// TIA Portal V20 export
DATA_BLOCK "ShiftmodelInterfaceHmi"   // DB103
TITLE = Schichtzeiten / ShiftmodelTimes
AUTHOR : SICAR
FAMILY : Shiftmodel
VERSION : 1.0
// Global DB fuer Schnittstelle HMI / Global DB for HMI interface
// stored: InstanceOfName LSicar_typeShiftmodelHmi, InstanceOfType UDT
"LSicar_typeShiftmodelHmi"
   // VAR RETAIN
   //    shiftTimesListIndex : DInt := 1;
   //    actualTimesDay : Array[0..7] of "LSicar_typeShiftmodTime1Day";
   //    actualSignalsDay : Array[0..7] of "LSicar_typeShiftmodSign1Day";
   //    summary : "LSicar_typeShiftmodSumHmi";
   //    actualDay : USInt := 0;
   //    shiftTimesListOnOff : Bool := TRUE;   // Schichtzeiten Remote OnOff / Shift times OnOff
   //    setAdjTimes : Bool := FALSE;
   //    hmiTimesValidFor : Array[0..3] of "LSicar_typeWeekdayBools";
   //    hmiTimes : Array[0..3] of "LSicar_typeShiftmodTime1Shift";   // Schnittstelle Lokale Zeiten (eingeben am HMI) / Interface Local Times (Input on HMI)
   //    productionTimes : "LSicar_typeProdTimesHmi";
   // END_VAR
BEGIN
   actualTimesDay[0].shift[0..3].endCircuitTime := TOD#00:00:00;
   actualTimesDay[1].shift[0..3].endCircuitTime := TOD#00:00:00;
   actualTimesDay[2].shift[0..3].endCircuitTime := TOD#00:00:00;
   actualTimesDay[3].shift[0..3].endCircuitTime := TOD#00:00:00;
   actualTimesDay[4].shift[0..3].endCircuitTime := TOD#00:00:00;
   actualTimesDay[5].shift[0..3].endCircuitTime := TOD#00:00:00;
   actualTimesDay[6].shift[0..3].endCircuitTime := TOD#00:00:00;
   actualTimesDay[7].shift[0..3].endCircuitTime := TOD#00:00:00;
   actualTimesDay[0].shift[0..3].start := TOD#00:00:00;
   actualTimesDay[1].shift[0..3].start := TOD#00:00:00;
   actualTimesDay[2].shift[0..3].start := TOD#00:00:00;
   actualTimesDay[3].shift[0..3].start := TOD#00:00:00;
   actualTimesDay[4].shift[0..3].start := TOD#00:00:00;
   actualTimesDay[5].shift[0..3].start := TOD#00:00:00;
   actualTimesDay[6].shift[0..3].start := TOD#00:00:00;
   actualTimesDay[7].shift[0..3].start := TOD#00:00:00;
   actualTimesDay[0].shift[0].break[0..4].start := TOD#00:00:00;
   actualTimesDay[0].shift[1].break[0..4].start := TOD#00:00:00;
   actualTimesDay[0].shift[2].break[0..4].start := TOD#00:00:00;
   actualTimesDay[0].shift[3].break[0..4].start := TOD#00:00:00;
   actualTimesDay[1].shift[0].break[0..4].start := TOD#00:00:00;
   actualTimesDay[1].shift[1].break[0..4].start := TOD#00:00:00;
   actualTimesDay[1].shift[2].break[0..4].start := TOD#00:00:00;
   actualTimesDay[1].shift[3].break[0..4].start := TOD#00:00:00;
   actualTimesDay[2].shift[0].break[0..4].start := TOD#00:00:00;
   actualTimesDay[2].shift[1].break[0..4].start := TOD#00:00:00;
   actualTimesDay[2].shift[2].break[0..4].start := TOD#00:00:00;
   actualTimesDay[2].shift[3].break[0..4].start := TOD#00:00:00;
   actualTimesDay[3].shift[0].break[0..4].start := TOD#00:00:00;
   actualTimesDay[3].shift[1].break[0..4].start := TOD#00:00:00;
   actualTimesDay[3].shift[2].break[0..4].start := TOD#00:00:00;
   actualTimesDay[3].shift[3].break[0..4].start := TOD#00:00:00;
   actualTimesDay[4].shift[0].break[0..4].start := TOD#00:00:00;
   actualTimesDay[4].shift[1].break[0..4].start := TOD#00:00:00;
   actualTimesDay[4].shift[2].break[0..4].start := TOD#00:00:00;
   actualTimesDay[4].shift[3].break[0..4].start := TOD#00:00:00;
   actualTimesDay[5].shift[0].break[0..4].start := TOD#00:00:00;
   actualTimesDay[5].shift[1].break[0..4].start := TOD#00:00:00;
   actualTimesDay[5].shift[2].break[0..4].start := TOD#00:00:00;
   actualTimesDay[5].shift[3].break[0..4].start := TOD#00:00:00;
   actualTimesDay[6].shift[0].break[0..4].start := TOD#00:00:00;
   actualTimesDay[6].shift[1].break[0..4].start := TOD#00:00:00;
   actualTimesDay[6].shift[2].break[0..4].start := TOD#00:00:00;
   actualTimesDay[6].shift[3].break[0..4].start := TOD#00:00:00;
   actualTimesDay[7].shift[0].break[0..4].start := TOD#00:00:00;
   actualTimesDay[7].shift[1].break[0..4].start := TOD#00:00:00;
   actualTimesDay[7].shift[2].break[0..4].start := TOD#00:00:00;
   actualTimesDay[7].shift[3].break[0..4].start := TOD#00:00:00;
   actualTimesDay[0].shift[0].break[0..4].startCircuitTime := TOD#00:00:00;
   actualTimesDay[0].shift[1].break[0..4].startCircuitTime := TOD#00:00:00;
   actualTimesDay[0].shift[2].break[0..4].startCircuitTime := TOD#00:00:00;
   actualTimesDay[0].shift[3].break[0..4].startCircuitTime := TOD#00:00:00;
   actualTimesDay[1].shift[0].break[0..4].startCircuitTime := TOD#00:00:00;
   actualTimesDay[1].shift[1].break[0..4].startCircuitTime := TOD#00:00:00;
   actualTimesDay[1].shift[2].break[0..4].startCircuitTime := TOD#00:00:00;
   actualTimesDay[1].shift[3].break[0..4].startCircuitTime := TOD#00:00:00;
   actualTimesDay[2].shift[0].break[0..4].startCircuitTime := TOD#00:00:00;
   actualTimesDay[2].shift[1].break[0..4].startCircuitTime := TOD#00:00:00;
   actualTimesDay[2].shift[2].break[0..4].startCircuitTime := TOD#00:00:00;
   actualTimesDay[2].shift[3].break[0..4].startCircuitTime := TOD#00:00:00;
   actualTimesDay[3].shift[0].break[0..4].startCircuitTime := TOD#00:00:00;
   actualTimesDay[3].shift[1].break[0..4].startCircuitTime := TOD#00:00:00;
   actualTimesDay[3].shift[2].break[0..4].startCircuitTime := TOD#00:00:00;
   actualTimesDay[3].shift[3].break[0..4].startCircuitTime := TOD#00:00:00;
   actualTimesDay[4].shift[0].break[0..4].startCircuitTime := TOD#00:00:00;
   actualTimesDay[4].shift[1].break[0..4].startCircuitTime := TOD#00:00:00;
   actualTimesDay[4].shift[2].break[0..4].startCircuitTime := TOD#00:00:00;
   actualTimesDay[4].shift[3].break[0..4].startCircuitTime := TOD#00:00:00;
   actualTimesDay[5].shift[0].break[0..4].startCircuitTime := TOD#00:00:00;
   actualTimesDay[5].shift[1].break[0..4].startCircuitTime := TOD#00:00:00;
   actualTimesDay[5].shift[2].break[0..4].startCircuitTime := TOD#00:00:00;
   actualTimesDay[5].shift[3].break[0..4].startCircuitTime := TOD#00:00:00;
   actualTimesDay[6].shift[0].break[0..4].startCircuitTime := TOD#00:00:00;
   actualTimesDay[6].shift[1].break[0..4].startCircuitTime := TOD#00:00:00;
   actualTimesDay[6].shift[2].break[0..4].startCircuitTime := TOD#00:00:00;
   actualTimesDay[6].shift[3].break[0..4].startCircuitTime := TOD#00:00:00;
   actualTimesDay[7].shift[0].break[0..4].startCircuitTime := TOD#00:00:00;
   actualTimesDay[7].shift[1].break[0..4].startCircuitTime := TOD#00:00:00;
   actualTimesDay[7].shift[2].break[0..4].startCircuitTime := TOD#00:00:00;
   actualTimesDay[7].shift[3].break[0..4].startCircuitTime := TOD#00:00:00;
   actualTimesDay[0].shift[0].break[0..4].endCircuitTime := TOD#00:00:00;
   actualTimesDay[0].shift[1].break[0..4].endCircuitTime := TOD#00:00:00;
   actualTimesDay[0].shift[2].break[0..4].endCircuitTime := TOD#00:00:00;
   actualTimesDay[0].shift[3].break[0..4].endCircuitTime := TOD#00:00:00;
   actualTimesDay[1].shift[0].break[0..4].endCircuitTime := TOD#00:00:00;
   actualTimesDay[1].shift[1].break[0..4].endCircuitTime := TOD#00:00:00;
   actualTimesDay[1].shift[2].break[0..4].endCircuitTime := TOD#00:00:00;
   actualTimesDay[1].shift[3].break[0..4].endCircuitTime := TOD#00:00:00;
   actualTimesDay[2].shift[0].break[0..4].endCircuitTime := TOD#00:00:00;
   actualTimesDay[2].shift[1].break[0..4].endCircuitTime := TOD#00:00:00;
   actualTimesDay[2].shift[2].break[0..4].endCircuitTime := TOD#00:00:00;
   actualTimesDay[2].shift[3].break[0..4].endCircuitTime := TOD#00:00:00;
   actualTimesDay[3].shift[0].break[0..4].endCircuitTime := TOD#00:00:00;
   actualTimesDay[3].shift[1].break[0..4].endCircuitTime := TOD#00:00:00;
   actualTimesDay[3].shift[2].break[0..4].endCircuitTime := TOD#00:00:00;
   actualTimesDay[3].shift[3].break[0..4].endCircuitTime := TOD#00:00:00;
   actualTimesDay[4].shift[0].break[0..4].endCircuitTime := TOD#00:00:00;
   actualTimesDay[4].shift[1].break[0..4].endCircuitTime := TOD#00:00:00;
   actualTimesDay[4].shift[2].break[0..4].endCircuitTime := TOD#00:00:00;
   actualTimesDay[4].shift[3].break[0..4].endCircuitTime := TOD#00:00:00;
   actualTimesDay[5].shift[0].break[0..4].endCircuitTime := TOD#00:00:00;
   actualTimesDay[5].shift[1].break[0..4].endCircuitTime := TOD#00:00:00;
   actualTimesDay[5].shift[2].break[0..4].endCircuitTime := TOD#00:00:00;
   actualTimesDay[5].shift[3].break[0..4].endCircuitTime := TOD#00:00:00;
   actualTimesDay[6].shift[0].break[0..4].endCircuitTime := TOD#00:00:00;
   actualTimesDay[6].shift[1].break[0..4].endCircuitTime := TOD#00:00:00;
   actualTimesDay[6].shift[2].break[0..4].endCircuitTime := TOD#00:00:00;
   actualTimesDay[6].shift[3].break[0..4].endCircuitTime := TOD#00:00:00;
   actualTimesDay[7].shift[0].break[0..4].endCircuitTime := TOD#00:00:00;
   actualTimesDay[7].shift[1].break[0..4].endCircuitTime := TOD#00:00:00;
   actualTimesDay[7].shift[2].break[0..4].endCircuitTime := TOD#00:00:00;
   actualTimesDay[7].shift[3].break[0..4].endCircuitTime := TOD#00:00:00;
   actualTimesDay[0].shift[0].break[0..4].end := TOD#00:00:00;
   actualTimesDay[0].shift[1].break[0..4].end := TOD#00:00:00;
   actualTimesDay[0].shift[2].break[0..4].end := TOD#00:00:00;
   actualTimesDay[0].shift[3].break[0..4].end := TOD#00:00:00;
   actualTimesDay[1].shift[0].break[0..4].end := TOD#00:00:00;
   actualTimesDay[1].shift[1].break[0..4].end := TOD#00:00:00;
   actualTimesDay[1].shift[2].break[0..4].end := TOD#00:00:00;
   actualTimesDay[1].shift[3].break[0..4].end := TOD#00:00:00;
   actualTimesDay[2].shift[0].break[0..4].end := TOD#00:00:00;
   actualTimesDay[2].shift[1].break[0..4].end := TOD#00:00:00;
   actualTimesDay[2].shift[2].break[0..4].end := TOD#00:00:00;
   actualTimesDay[2].shift[3].break[0..4].end := TOD#00:00:00;
   actualTimesDay[3].shift[0].break[0..4].end := TOD#00:00:00;
   actualTimesDay[3].shift[1].break[0..4].end := TOD#00:00:00;
   actualTimesDay[3].shift[2].break[0..4].end := TOD#00:00:00;
   actualTimesDay[3].shift[3].break[0..4].end := TOD#00:00:00;
   actualTimesDay[4].shift[0].break[0..4].end := TOD#00:00:00;
   actualTimesDay[4].shift[1].break[0..4].end := TOD#00:00:00;
   actualTimesDay[4].shift[2].break[0..4].end := TOD#00:00:00;
   actualTimesDay[4].shift[3].break[0..4].end := TOD#00:00:00;
   actualTimesDay[5].shift[0].break[0..4].end := TOD#00:00:00;
   actualTimesDay[5].shift[1].break[0..4].end := TOD#00:00:00;
   actualTimesDay[5].shift[2].break[0..4].end := TOD#00:00:00;
   actualTimesDay[5].shift[3].break[0..4].end := TOD#00:00:00;
   actualTimesDay[6].shift[0].break[0..4].end := TOD#00:00:00;
   actualTimesDay[6].shift[1].break[0..4].end := TOD#00:00:00;
   actualTimesDay[6].shift[2].break[0..4].end := TOD#00:00:00;
   actualTimesDay[6].shift[3].break[0..4].end := TOD#00:00:00;
   actualTimesDay[7].shift[0].break[0..4].end := TOD#00:00:00;
   actualTimesDay[7].shift[1].break[0..4].end := TOD#00:00:00;
   actualTimesDay[7].shift[2].break[0..4].end := TOD#00:00:00;
   actualTimesDay[7].shift[3].break[0..4].end := TOD#00:00:00;
   actualTimesDay[0].shift[0..3].end := TOD#00:00:00;
   actualTimesDay[1].shift[0..3].end := TOD#00:00:00;
   actualTimesDay[2].shift[0..3].end := TOD#00:00:00;
   actualTimesDay[3].shift[0..3].end := TOD#00:00:00;
   actualTimesDay[4].shift[0..3].end := TOD#00:00:00;
   actualTimesDay[5].shift[0..3].end := TOD#00:00:00;
   actualTimesDay[6].shift[0..3].end := TOD#00:00:00;
   actualTimesDay[7].shift[0..3].end := TOD#00:00:00;
   actualTimesDay[0].shift[0..3].startCircuitTime := TOD#00:00:00;
   actualTimesDay[1].shift[0..3].startCircuitTime := TOD#00:00:00;
   actualTimesDay[2].shift[0..3].startCircuitTime := TOD#00:00:00;
   actualTimesDay[3].shift[0..3].startCircuitTime := TOD#00:00:00;
   actualTimesDay[4].shift[0..3].startCircuitTime := TOD#00:00:00;
   actualTimesDay[5].shift[0..3].startCircuitTime := TOD#00:00:00;
   actualTimesDay[6].shift[0..3].startCircuitTime := TOD#00:00:00;
   actualTimesDay[7].shift[0..3].startCircuitTime := TOD#00:00:00;
   actualSignalsDay[0].shift[0..3].shiftConfig := FALSE;
   actualSignalsDay[1].shift[0..3].shiftConfig := FALSE;
   actualSignalsDay[2].shift[0..3].shiftConfig := FALSE;
   actualSignalsDay[3].shift[0..3].shiftConfig := FALSE;
   actualSignalsDay[4].shift[0..3].shiftConfig := FALSE;
   actualSignalsDay[5].shift[0..3].shiftConfig := FALSE;
   actualSignalsDay[6].shift[0..3].shiftConfig := FALSE;
   actualSignalsDay[7].shift[0..3].shiftConfig := FALSE;
   actualSignalsDay[0].shift[0..3].shiftActive := FALSE;
   actualSignalsDay[1].shift[0..3].shiftActive := FALSE;
   actualSignalsDay[2].shift[0..3].shiftActive := FALSE;
   actualSignalsDay[3].shift[0..3].shiftActive := FALSE;
   actualSignalsDay[4].shift[0..3].shiftActive := FALSE;
   actualSignalsDay[5].shift[0..3].shiftActive := FALSE;
   actualSignalsDay[6].shift[0..3].shiftActive := FALSE;
   actualSignalsDay[7].shift[0..3].shiftActive := FALSE;
   actualSignalsDay[0].shift[0..3].shiftEndCirTimeConfig := FALSE;
   actualSignalsDay[1].shift[0..3].shiftEndCirTimeConfig := FALSE;
   actualSignalsDay[2].shift[0..3].shiftEndCirTimeConfig := FALSE;
   actualSignalsDay[3].shift[0..3].shiftEndCirTimeConfig := FALSE;
   actualSignalsDay[4].shift[0..3].shiftEndCirTimeConfig := FALSE;
   actualSignalsDay[5].shift[0..3].shiftEndCirTimeConfig := FALSE;
   actualSignalsDay[6].shift[0..3].shiftEndCirTimeConfig := FALSE;
   actualSignalsDay[7].shift[0..3].shiftEndCirTimeConfig := FALSE;
   actualSignalsDay[0].shift[0..3].shiftStartCirTimeConfig := FALSE;
   actualSignalsDay[1].shift[0..3].shiftStartCirTimeConfig := FALSE;
   actualSignalsDay[2].shift[0..3].shiftStartCirTimeConfig := FALSE;
   actualSignalsDay[3].shift[0..3].shiftStartCirTimeConfig := FALSE;
   actualSignalsDay[4].shift[0..3].shiftStartCirTimeConfig := FALSE;
   actualSignalsDay[5].shift[0..3].shiftStartCirTimeConfig := FALSE;
   actualSignalsDay[6].shift[0..3].shiftStartCirTimeConfig := FALSE;
   actualSignalsDay[7].shift[0..3].shiftStartCirTimeConfig := FALSE;
   actualSignalsDay[0].shift[0..3].shiftEndCirTimeActive := FALSE;
   actualSignalsDay[1].shift[0..3].shiftEndCirTimeActive := FALSE;
   actualSignalsDay[2].shift[0..3].shiftEndCirTimeActive := FALSE;
   actualSignalsDay[3].shift[0..3].shiftEndCirTimeActive := FALSE;
   actualSignalsDay[4].shift[0..3].shiftEndCirTimeActive := FALSE;
   actualSignalsDay[5].shift[0..3].shiftEndCirTimeActive := FALSE;
   actualSignalsDay[6].shift[0..3].shiftEndCirTimeActive := FALSE;
   actualSignalsDay[7].shift[0..3].shiftEndCirTimeActive := FALSE;
   actualSignalsDay[0].shift[0..3].shiftStartCirTimeActive := FALSE;
   actualSignalsDay[1].shift[0..3].shiftStartCirTimeActive := FALSE;
   actualSignalsDay[2].shift[0..3].shiftStartCirTimeActive := FALSE;
   actualSignalsDay[3].shift[0..3].shiftStartCirTimeActive := FALSE;
   actualSignalsDay[4].shift[0..3].shiftStartCirTimeActive := FALSE;
   actualSignalsDay[5].shift[0..3].shiftStartCirTimeActive := FALSE;
   actualSignalsDay[6].shift[0..3].shiftStartCirTimeActive := FALSE;
   actualSignalsDay[7].shift[0..3].shiftStartCirTimeActive := FALSE;
   actualSignalsDay[0].shift[0..3].shiftSignalsHmi := 16#00;
   actualSignalsDay[1].shift[0..3].shiftSignalsHmi := 16#00;
   actualSignalsDay[2].shift[0..3].shiftSignalsHmi := 16#00;
   actualSignalsDay[3].shift[0..3].shiftSignalsHmi := 16#00;
   actualSignalsDay[4].shift[0..3].shiftSignalsHmi := 16#00;
   actualSignalsDay[5].shift[0..3].shiftSignalsHmi := 16#00;
   actualSignalsDay[6].shift[0..3].shiftSignalsHmi := 16#00;
   actualSignalsDay[7].shift[0..3].shiftSignalsHmi := 16#00;
   actualSignalsDay[0].shift[0].break[0..4].config := FALSE;
   actualSignalsDay[0].shift[1].break[0..4].config := FALSE;
   actualSignalsDay[0].shift[2].break[0..4].config := FALSE;
   actualSignalsDay[0].shift[3].break[0..4].config := FALSE;
   actualSignalsDay[1].shift[0].break[0..4].config := FALSE;
   actualSignalsDay[1].shift[1].break[0..4].config := FALSE;
   actualSignalsDay[1].shift[2].break[0..4].config := FALSE;
   actualSignalsDay[1].shift[3].break[0..4].config := FALSE;
   actualSignalsDay[2].shift[0].break[0..4].config := FALSE;
   actualSignalsDay[2].shift[1].break[0..4].config := FALSE;
   actualSignalsDay[2].shift[2].break[0..4].config := FALSE;
   actualSignalsDay[2].shift[3].break[0..4].config := FALSE;
   actualSignalsDay[3].shift[0].break[0..4].config := FALSE;
   actualSignalsDay[3].shift[1].break[0..4].config := FALSE;
   actualSignalsDay[3].shift[2].break[0..4].config := FALSE;
   actualSignalsDay[3].shift[3].break[0..4].config := FALSE;
   actualSignalsDay[4].shift[0].break[0..4].config := FALSE;
   actualSignalsDay[4].shift[1].break[0..4].config := FALSE;
   actualSignalsDay[4].shift[2].break[0..4].config := FALSE;
   actualSignalsDay[4].shift[3].break[0..4].config := FALSE;
   actualSignalsDay[5].shift[0].break[0..4].config := FALSE;
   actualSignalsDay[5].shift[1].break[0..4].config := FALSE;
   actualSignalsDay[5].shift[2].break[0..4].config := FALSE;
   actualSignalsDay[5].shift[3].break[0..4].config := FALSE;
   actualSignalsDay[6].shift[0].break[0..4].config := FALSE;
   actualSignalsDay[6].shift[1].break[0..4].config := FALSE;
   actualSignalsDay[6].shift[2].break[0..4].config := FALSE;
   actualSignalsDay[6].shift[3].break[0..4].config := FALSE;
   actualSignalsDay[7].shift[0].break[0..4].config := FALSE;
   actualSignalsDay[7].shift[1].break[0..4].config := FALSE;
   actualSignalsDay[7].shift[2].break[0..4].config := FALSE;
   actualSignalsDay[7].shift[3].break[0..4].config := FALSE;
   actualSignalsDay[0].shift[0].break[0..4].active := FALSE;
   actualSignalsDay[0].shift[1].break[0..4].active := FALSE;
   actualSignalsDay[0].shift[2].break[0..4].active := FALSE;
   actualSignalsDay[0].shift[3].break[0..4].active := FALSE;
   actualSignalsDay[1].shift[0].break[0..4].active := FALSE;
   actualSignalsDay[1].shift[1].break[0..4].active := FALSE;
   actualSignalsDay[1].shift[2].break[0..4].active := FALSE;
   actualSignalsDay[1].shift[3].break[0..4].active := FALSE;
   actualSignalsDay[2].shift[0].break[0..4].active := FALSE;
   actualSignalsDay[2].shift[1].break[0..4].active := FALSE;
   actualSignalsDay[2].shift[2].break[0..4].active := FALSE;
   actualSignalsDay[2].shift[3].break[0..4].active := FALSE;
   actualSignalsDay[3].shift[0].break[0..4].active := FALSE;
   actualSignalsDay[3].shift[1].break[0..4].active := FALSE;
   actualSignalsDay[3].shift[2].break[0..4].active := FALSE;
   actualSignalsDay[3].shift[3].break[0..4].active := FALSE;
   actualSignalsDay[4].shift[0].break[0..4].active := FALSE;
   actualSignalsDay[4].shift[1].break[0..4].active := FALSE;
   actualSignalsDay[4].shift[2].break[0..4].active := FALSE;
   actualSignalsDay[4].shift[3].break[0..4].active := FALSE;
   actualSignalsDay[5].shift[0].break[0..4].active := FALSE;
   actualSignalsDay[5].shift[1].break[0..4].active := FALSE;
   actualSignalsDay[5].shift[2].break[0..4].active := FALSE;
   actualSignalsDay[5].shift[3].break[0..4].active := FALSE;
   actualSignalsDay[6].shift[0].break[0..4].active := FALSE;
   actualSignalsDay[6].shift[1].break[0..4].active := FALSE;
   actualSignalsDay[6].shift[2].break[0..4].active := FALSE;
   actualSignalsDay[6].shift[3].break[0..4].active := FALSE;
   actualSignalsDay[7].shift[0].break[0..4].active := FALSE;
   actualSignalsDay[7].shift[1].break[0..4].active := FALSE;
   actualSignalsDay[7].shift[2].break[0..4].active := FALSE;
   actualSignalsDay[7].shift[3].break[0..4].active := FALSE;
   actualSignalsDay[0].shift[0].break[0..4].circuitTimeConfig := FALSE;
   actualSignalsDay[0].shift[1].break[0..4].circuitTimeConfig := FALSE;
   actualSignalsDay[0].shift[2].break[0..4].circuitTimeConfig := FALSE;
   actualSignalsDay[0].shift[3].break[0..4].circuitTimeConfig := FALSE;
   actualSignalsDay[1].shift[0].break[0..4].circuitTimeConfig := FALSE;
   actualSignalsDay[1].shift[1].break[0..4].circuitTimeConfig := FALSE;
   actualSignalsDay[1].shift[2].break[0..4].circuitTimeConfig := FALSE;
   actualSignalsDay[1].shift[3].break[0..4].circuitTimeConfig := FALSE;
   actualSignalsDay[2].shift[0].break[0..4].circuitTimeConfig := FALSE;
   actualSignalsDay[2].shift[1].break[0..4].circuitTimeConfig := FALSE;
   actualSignalsDay[2].shift[2].break[0..4].circuitTimeConfig := FALSE;
   actualSignalsDay[2].shift[3].break[0..4].circuitTimeConfig := FALSE;
   actualSignalsDay[3].shift[0].break[0..4].circuitTimeConfig := FALSE;
   actualSignalsDay[3].shift[1].break[0..4].circuitTimeConfig := FALSE;
   actualSignalsDay[3].shift[2].break[0..4].circuitTimeConfig := FALSE;
   actualSignalsDay[3].shift[3].break[0..4].circuitTimeConfig := FALSE;
   actualSignalsDay[4].shift[0].break[0..4].circuitTimeConfig := FALSE;
   actualSignalsDay[4].shift[1].break[0..4].circuitTimeConfig := FALSE;
   actualSignalsDay[4].shift[2].break[0..4].circuitTimeConfig := FALSE;
   actualSignalsDay[4].shift[3].break[0..4].circuitTimeConfig := FALSE;
   actualSignalsDay[5].shift[0].break[0..4].circuitTimeConfig := FALSE;
   actualSignalsDay[5].shift[1].break[0..4].circuitTimeConfig := FALSE;
   actualSignalsDay[5].shift[2].break[0..4].circuitTimeConfig := FALSE;
   actualSignalsDay[5].shift[3].break[0..4].circuitTimeConfig := FALSE;
   actualSignalsDay[6].shift[0].break[0..4].circuitTimeConfig := FALSE;
   actualSignalsDay[6].shift[1].break[0..4].circuitTimeConfig := FALSE;
   actualSignalsDay[6].shift[2].break[0..4].circuitTimeConfig := FALSE;
   actualSignalsDay[6].shift[3].break[0..4].circuitTimeConfig := FALSE;
   actualSignalsDay[7].shift[0].break[0..4].circuitTimeConfig := FALSE;
   actualSignalsDay[7].shift[1].break[0..4].circuitTimeConfig := FALSE;
   actualSignalsDay[7].shift[2].break[0..4].circuitTimeConfig := FALSE;
   actualSignalsDay[7].shift[3].break[0..4].circuitTimeConfig := FALSE;
   actualSignalsDay[0].shift[0].break[0..4].circuitTimeActive := FALSE;
   actualSignalsDay[0].shift[1].break[0..4].circuitTimeActive := FALSE;
   actualSignalsDay[0].shift[2].break[0..4].circuitTimeActive := FALSE;
   actualSignalsDay[0].shift[3].break[0..4].circuitTimeActive := FALSE;
   actualSignalsDay[1].shift[0].break[0..4].circuitTimeActive := FALSE;
   actualSignalsDay[1].shift[1].break[0..4].circuitTimeActive := FALSE;
   actualSignalsDay[1].shift[2].break[0..4].circuitTimeActive := FALSE;
   actualSignalsDay[1].shift[3].break[0..4].circuitTimeActive := FALSE;
   actualSignalsDay[2].shift[0].break[0..4].circuitTimeActive := FALSE;
   actualSignalsDay[2].shift[1].break[0..4].circuitTimeActive := FALSE;
   actualSignalsDay[2].shift[2].break[0..4].circuitTimeActive := FALSE;
   actualSignalsDay[2].shift[3].break[0..4].circuitTimeActive := FALSE;
   actualSignalsDay[3].shift[0].break[0..4].circuitTimeActive := FALSE;
   actualSignalsDay[3].shift[1].break[0..4].circuitTimeActive := FALSE;
   actualSignalsDay[3].shift[2].break[0..4].circuitTimeActive := FALSE;
   actualSignalsDay[3].shift[3].break[0..4].circuitTimeActive := FALSE;
   actualSignalsDay[4].shift[0].break[0..4].circuitTimeActive := FALSE;
   actualSignalsDay[4].shift[1].break[0..4].circuitTimeActive := FALSE;
   actualSignalsDay[4].shift[2].break[0..4].circuitTimeActive := FALSE;
   actualSignalsDay[4].shift[3].break[0..4].circuitTimeActive := FALSE;
   actualSignalsDay[5].shift[0].break[0..4].circuitTimeActive := FALSE;
   actualSignalsDay[5].shift[1].break[0..4].circuitTimeActive := FALSE;
   actualSignalsDay[5].shift[2].break[0..4].circuitTimeActive := FALSE;
   actualSignalsDay[5].shift[3].break[0..4].circuitTimeActive := FALSE;
   actualSignalsDay[6].shift[0].break[0..4].circuitTimeActive := FALSE;
   actualSignalsDay[6].shift[1].break[0..4].circuitTimeActive := FALSE;
   actualSignalsDay[6].shift[2].break[0..4].circuitTimeActive := FALSE;
   actualSignalsDay[6].shift[3].break[0..4].circuitTimeActive := FALSE;
   actualSignalsDay[7].shift[0].break[0..4].circuitTimeActive := FALSE;
   actualSignalsDay[7].shift[1].break[0..4].circuitTimeActive := FALSE;
   actualSignalsDay[7].shift[2].break[0..4].circuitTimeActive := FALSE;
   actualSignalsDay[7].shift[3].break[0..4].circuitTimeActive := FALSE;
   actualSignalsDay[0].shift[0..3].breakSignalsHmi := 16#0000;
   actualSignalsDay[1].shift[0..3].breakSignalsHmi := 16#0000;
   actualSignalsDay[2].shift[0..3].breakSignalsHmi := 16#0000;
   actualSignalsDay[3].shift[0..3].breakSignalsHmi := 16#0000;
   actualSignalsDay[4].shift[0..3].breakSignalsHmi := 16#0000;
   actualSignalsDay[5].shift[0..3].breakSignalsHmi := 16#0000;
   actualSignalsDay[6].shift[0..3].breakSignalsHmi := 16#0000;
   actualSignalsDay[7].shift[0..3].breakSignalsHmi := 16#0000;
   actualSignalsDay[0..7].shiftsPerDay := 0;
   summary.earlyShiftActive := FALSE;
   summary.lateShiftActive := FALSE;
   summary.nightShiftActive := FALSE;
   summary.breakInShiftActive := FALSE;
   summary.breakBetweenShiftAct := FALSE;
   summary.breakActive := FALSE;
   summary.circuitTimeInShiftAct := FALSE;
   summary.circuitTimeBetwShiftAct := FALSE;
   summary.circuitTimeActive := FALSE;
   summary.noOfWorkdays := 0;
   summary.workdays[0..7] := FALSE;
   hmiTimesValidFor[0..3].sunday := FALSE;
   hmiTimesValidFor[0..3].monday := FALSE;
   hmiTimesValidFor[0..3].tuesday := FALSE;
   hmiTimesValidFor[0..3].wednesday := FALSE;
   hmiTimesValidFor[0..3].thursday := FALSE;
   hmiTimesValidFor[0..3].friday := FALSE;
   hmiTimesValidFor[0..3].saturday := FALSE;
   hmiTimes[0].endCircuitTime := TOD#00:00:00;
   hmiTimes[1].endCircuitTime := TOD#05:57:00;
   hmiTimes[2].endCircuitTime := TOD#13:57:00;
   hmiTimes[3].endCircuitTime := TOD#21:57:00;
   hmiTimes[0].start := TOD#00:00:00;
   hmiTimes[1].start := TOD#06:00:00;
   hmiTimes[2].start := TOD#14:00:00;
   hmiTimes[3].start := TOD#22:00:00;
   hmiTimes[0].break[0..4].start := TOD#00:00:00;
   hmiTimes[1].break[0].start := TOD#00:00:00;
   hmiTimes[1].break[1].start := TOD#08:00:00;
   hmiTimes[1].break[2].start := TOD#10:00:00;
   hmiTimes[1].break[3].start := TOD#12:00:00;
   hmiTimes[1].break[4].start := TOD#00:00:00;
   hmiTimes[2].break[0].start := TOD#00:00:00;
   hmiTimes[2].break[1].start := TOD#16:00:00;
   hmiTimes[2].break[2].start := TOD#18:00:00;
   hmiTimes[2].break[3].start := TOD#20:00:00;
   hmiTimes[2].break[4].start := TOD#00:00:00;
   hmiTimes[3].break[0..1].start := TOD#00:00:00;
   hmiTimes[3].break[2].start := TOD#02:00:00;
   hmiTimes[3].break[3].start := TOD#04:00:00;
   hmiTimes[3].break[4].start := TOD#00:00:00;
   hmiTimes[0].break[0..4].startCircuitTime := TOD#00:00:00;
   hmiTimes[1].break[0].startCircuitTime := TOD#00:00:00;
   hmiTimes[1].break[1].startCircuitTime := TOD#08:02:00;
   hmiTimes[1].break[2].startCircuitTime := TOD#00:00:00;
   hmiTimes[1].break[3].startCircuitTime := TOD#12:02:00;
   hmiTimes[1].break[4].startCircuitTime := TOD#00:00:00;
   hmiTimes[2].break[0].startCircuitTime := TOD#00:00:00;
   hmiTimes[2].break[1].startCircuitTime := TOD#16:02:00;
   hmiTimes[2].break[2].startCircuitTime := TOD#00:00:00;
   hmiTimes[2].break[3].startCircuitTime := TOD#20:02:00;
   hmiTimes[2].break[4].startCircuitTime := TOD#00:00:00;
   hmiTimes[3].break[0].startCircuitTime := TOD#00:00:00;
   hmiTimes[3].break[1].startCircuitTime := TOD#00:02:00;
   hmiTimes[3].break[2].startCircuitTime := TOD#00:00:00;
   hmiTimes[3].break[3].startCircuitTime := TOD#04:02:00;
   hmiTimes[3].break[4].startCircuitTime := TOD#00:00:00;
   hmiTimes[0].break[0..4].endCircuitTime := TOD#00:00:00;
   hmiTimes[1].break[0].endCircuitTime := TOD#00:00:00;
   hmiTimes[1].break[1].endCircuitTime := TOD#08:13:00;
   hmiTimes[1].break[2].endCircuitTime := TOD#00:00:00;
   hmiTimes[1].break[3].endCircuitTime := TOD#12:13:00;
   hmiTimes[1].break[4].endCircuitTime := TOD#00:00:00;
   hmiTimes[2].break[0].endCircuitTime := TOD#00:00:00;
   hmiTimes[2].break[1].endCircuitTime := TOD#16:13:00;
   hmiTimes[2].break[2].endCircuitTime := TOD#00:00:00;
   hmiTimes[2].break[3].endCircuitTime := TOD#20:13:00;
   hmiTimes[2].break[4].endCircuitTime := TOD#00:00:00;
   hmiTimes[3].break[0].endCircuitTime := TOD#00:00:00;
   hmiTimes[3].break[1].endCircuitTime := TOD#00:13:00;
   hmiTimes[3].break[2].endCircuitTime := TOD#00:00:00;
   hmiTimes[3].break[3].endCircuitTime := TOD#04:13:00;
   hmiTimes[3].break[4].endCircuitTime := TOD#00:00:00;
   hmiTimes[0].break[0..4].end := TOD#00:00:00;
   hmiTimes[1].break[0].end := TOD#00:00:00;
   hmiTimes[1].break[1].end := TOD#08:15:00;
   hmiTimes[1].break[2].end := TOD#10:10:00;
   hmiTimes[1].break[3].end := TOD#12:15:00;
   hmiTimes[1].break[4].end := TOD#00:00:00;
   hmiTimes[2].break[0].end := TOD#00:00:00;
   hmiTimes[2].break[1].end := TOD#16:15:00;
   hmiTimes[2].break[2].end := TOD#18:10:00;
   hmiTimes[2].break[3].end := TOD#20:15:00;
   hmiTimes[2].break[4].end := TOD#00:00:00;
   hmiTimes[3].break[0].end := TOD#00:00:00;
   hmiTimes[3].break[1].end := TOD#00:15:00;
   hmiTimes[3].break[2].end := TOD#02:10:00;
   hmiTimes[3].break[3].end := TOD#04:15:00;
   hmiTimes[3].break[4].end := TOD#00:00:00;
   hmiTimes[0].end := TOD#00:00:00;
   hmiTimes[1].end := TOD#13:30:00;
   hmiTimes[2].end := TOD#21:30:00;
   hmiTimes[3].end := TOD#05:30:00;
   hmiTimes[0].startCircuitTime := TOD#00:00:00;
   hmiTimes[1].startCircuitTime := TOD#13:33:00;
   hmiTimes[2].startCircuitTime := TOD#21:33:00;
   hmiTimes[3].startCircuitTime := TOD#05:33:00;
   productionTimes.currentShiftTimes.start := TOD#00:00:00;
   productionTimes.currentShiftTimes.break[0..4].start := TOD#00:00:00;
   productionTimes.currentShiftTimes.break[0..4].startCircuitTime := TOD#00:00:00;
   productionTimes.currentShiftTimes.break[0..4].endCircuitTime := TOD#00:00:00;
   productionTimes.currentShiftTimes.break[0..4].end := TOD#00:00:00;
   productionTimes.currentShiftTimes.end := TOD#00:00:00;
   productionTimes.prodTimeTarget := TOD#00:00:00;
   productionTimes.prodTimeTargetTime := T#0MS;
   productionTimes.prodTimeExpired := TOD#00:00:00;
   productionTimes.prodTimeExpiredTime := T#0MS;
   productionTimes.breakActSum := FALSE;
   productionTimes.shiftActive := FALSE;
END_DATA_BLOCK
